# B&R Automation Studio project Embraco_LinkaNaOdlievanieRotorov_DokoncovaciaStanica_Rev2 (part 5)

#### Main.st - Init, cyclic, exit code
```iecst
PROGRAM _INIT
	MpRecipeXml_1.Load:= TRUE;
	ZvolenyUzivatel:= '';
	ZvolenaUroven:= 0;
	TP_ZobrazPopUpPrihlasenie:=1;

END_PROGRAM

PROGRAM _CYCLIC

	//Volanie funkcie SequenceControl//
	SequenceControl(SC:= SC_Uzivatelia);

	//Načítanie receptur z pamäte//
	IF MpRecipeXml_1.Load AND (MpRecipeXml_1.CommandDone OR MpRecipeXml_1.Error) THEN
		MpRecipeXml_1.Load:= FALSE;
		old_a:= 1;
		i:= 0;
		IndexZoznam:= 0;
	END_IF

	//Konfigurácia receptur//
	MpRecipeXml_1.MpLink:= ADR(gRecipeUzivatelXmlLink);  //takto sa menuje mapp komponenta v configurating view//
	MpRecipeXml_1.Enable:= TRUE;
	MpRecipeXml_1.Category:= ADR('UZIVATELIA');
	MpRecipeXml_1.Category:= ADR(strCategory);
	MpRecipeXml_1.DeviceName:= ADR('HDD');  //Názov media, kde sa budú receptury ukladat//
	MpRecipeXml_1.FileName:= ADR('UlozenyUzivatel'); //Názov súboru do ktorého sa receptúry uložia//
	MpRecipeXml_1();

	MpRecipeRegPar_1.MpLink:= ADR(gRecipeUzivatelXmlLink);
	MpRecipeRegPar_1.Enable:= TRUE;
	MpRecipeRegPar_1.Category:= ADR('UZIVATELIA');
	MpRecipeRegPar_1.PVName:= ADR('Uzivatel'); //Názov premenné, kde je vytvorená štruktura dat pre receptury//
	MpRecipeRegPar_1();

	//Zobrazenie názvou receptúr//
	FOR IndexZoznam:=0 TO 20 BY 1 DO
		ZoznamUzivatelov[IndexZoznam]:= Uzivatel[IndexZoznam].Meno;
	END_FOR

	//Posun indexu//
	IF MoveUP THEN
		IF i< 20 THEN
			i:= i+1;
		END_IF
		MoveUP:= FALSE;
	END_IF

	IF MoveDown THEN
		IF i>0 THEN
			i:= i-1;
		END_IF
		MoveDown:= FALSE;
	END_IF

	//Listovanie v uložených uživateloch//
	IF old_a <> i AND i >= 0 AND i <= 20 THEN
		MenoUzivatela:= Uzivatel[i].Meno;
		HesloUzivatela:= Uzivatel[i].Heslo;
		UrovenUzivatela:= Uzivatel[i].UrovenUzivatela;
		old_a:= i;
	END_IF

	//Prihlasovanie//
	CASE SC_Uzivatelia.Step OF

		0://Vynulovanie uživatela//
			SC_Uzivatelia.StepName:= '0 - Nulovanie';
			UlozUzivatelov:= FALSE;
			PrihlasUzivatela:= FALSE;
			VymazUzivatela:= FALSE;
			OdhlasUzivatela:= FALSE;
			MpRecipeXml_1.Save:= FALSE;
			b:= 0;
			SC_Uzivatelia.ResetStep:= TRUE;
			SC_Uzivatelia.Step:= 1;

		1://Rozhodnutie o činnosti//
			SC_Uzivatelia.StepName:= '1 - Rozhodnutie o cinnosti';
			IF UlozUzivatelov THEN
				SC_Uzivatelia.Step:= 10;
			ELSIF PrihlasUzivatela THEN
				SC_Uzivatelia.Step:= 20;
			ELSIF OdhlasUzivatela THEN
				SC_Uzivatelia.Step:= 30;
			ELSIF VymazUzivatela THEN
				SC_Uzivatelia.Step:= 40;
			END_IF

		10://Ulozenie uzivatela//
			SC_Uzivatelia.StepName:= '10 - Ulozenie uzivatela';
			Uzivatel[i].Meno:= MenoUzivatela;
			Uzivatel[i].Heslo:= HesloUzivatela;
			Uzivatel[i].UrovenUzivatela:= UrovenUzivatela;
			MpRecipeXml_1.Save:= TRUE;
			IF MpRecipeXml_1.CommandDone THEN
				SC_Uzivatelia.ResetStep:= TRUE;
				SC_Uzivatelia.Step:= 0;
			END_IF

		20://Čakanie na prihlásenie uživatela//
			SC_Uzivatelia.StepName:= '20 - Kontrola prazdneho uzivatela';
			IF ZadaneMenoUzivatela <> '' AND ZadaneHesloUzivatela <> '' THEN
				SC_Uzivatelia.ResetStep:= TRUE;
				SC_Uzivatelia.Step:= 21;
			ELSE
				ZadaneHesloUzivatela:= '';
				SC_Uzivatelia.ResetStep:= TRUE;
				SC_Uzivatelia.Step:= 0;
			END_IF

		21://Kontrola prihláseného uživatela//
			SC_Uzivatelia.StepName:= '21 - Kontrola prihláseného uzivatela';
			IF Uzivatel[b].Meno = ZadaneMenoUzivatela AND Uzivatel[b].Heslo = ZadaneHesloUzivatela THEN
				ZvolenyUzivatel:= Uzivatel[b].Meno;
				ZvolenaUroven:= Uzivatel[b].UrovenUzivatela;
				ZadaneHesloUzivatela:= '';
				SC_Uzivatelia.ResetStep:= TRUE;
				SC_Uzivatelia.Step:= 0;
			ELSE
				b:= b + 1;
				IF b = 21 OR b < 0 OR b > 21 THEN
					ZadaneMenoUzivatela:= '';
					ZadaneHesloUzivatela:= '';
					SC_Uzivatelia.ResetStep:= TRUE;
					SC_Uzivatelia.Step:= 0;
				END_IF
			END_IF

		30://Odhlásenie uživatela//
			SC_Uzivatelia.StepName:= '30 - Odhlasenie uzivatela';
			ZvolenyUzivatel:= '';
			ZvolenaUroven:= 0;
			SC_Uzivatelia.ResetStep:= TRUE;
			SC_Uzivatelia.Step:= 0;

		40://Vymazanie uživatela//
			SC_Uzivatelia.StepName:= '40 - Vymazanie uzivatela';
			Uzivatel[i].Meno:= '';
			Uzivatel[i].Heslo:= '';
			Uzivatel[i].UrovenUzivatela:= 0;
			MpRecipeXml_1.Save:= TRUE;
			IF MpRecipeXml_1.CommandDone THEN
				SC_Uzivatelia.ResetStep:= TRUE;
				SC_Uzivatelia.Step:= 0;
			END_IF

	END_CASE

END_PROGRAM

PROGRAM _EXIT
	(* Insert code here *)

END_PROGRAM
```

#### Variables.var - Local variables
```iecst
VAR
	strCategory : STRING[80];
	MpRecipeUI_1 : MpRecipeUI;
	UISetup : MpRecipeUISetupType;
	UIConnect : MpRecipeUIConnectType := (0);
	i : INT := 0;
	a : INT;
	old_a : INT := 0;
	MoveUP : BOOL;
	MoveDown : BOOL;
	IndexZoznam : INT;
	b : INT;
END_VAR
```

### Program Logical/Blikace/Blikanie1s (IEC)

#### Blikanie1s.st - Init, cyclic, exit code
```iecst
PROGRAM _INIT
	(* Insert code here *)

END_PROGRAM

PROGRAM _CYCLIC
	IF NOT Blikac1s THEN
		Blikac1s:= TRUE;
	ELSE
		Blikac1s:= FALSE;
	END_IF

END_PROGRAM

PROGRAM _EXIT
	(* Insert code here *)

END_PROGRAM
```

### Program Logical/Blikace/Blikanie200ms (IEC)

#### Blikanie200ms.st - Init, cyclic, exit code
```iecst
PROGRAM _INIT
	(* Insert code here *)

END_PROGRAM

PROGRAM _CYCLIC

	IF NOT Blikac200ms THEN
		Blikac200ms:= TRUE;
	ELSE
		Blikac200ms:= FALSE;
	END_IF

END_PROGRAM

PROGRAM _EXIT
	(* Insert code here *)

END_PROGRAM
```

### Program Logical/Blikace/Blikanie10ms (IEC)

#### Blikanie10ms.st - Init, cyclic, exit code
```iecst
PROGRAM _INIT
	(* Insert code here *)

END_PROGRAM

PROGRAM _CYCLIC
	IF NOT Blikac10ms THEN
		Blikac10ms:= TRUE;
	ELSE
		Blikac10ms:= FALSE;
	END_IF

END_PROGRAM

PROGRAM _EXIT
	(* Insert code here *)

END_PROGRAM
```

### Program Logical/Blikace/Blikanie50ms (IEC)

#### Blikanie50ms.st - Init, cyclic, exit code
```iecst
PROGRAM _INIT
	(* Insert code here *)

END_PROGRAM

PROGRAM _CYCLIC
	IF NOT Blikac50ms THEN
		Blikac50ms:= TRUE;
	ELSE
		Blikac50ms:= FALSE;
	END_IF

END_PROGRAM

PROGRAM _EXIT
	(* Insert code here *)

END_PROGRAM
```

### Program Logical/Blikace/Blikanie500ms (IEC)

#### Blikanie500ms.st - Init, cyclic, exit code
```iecst
PROGRAM _INIT
	(* Insert code here *)

END_PROGRAM

PROGRAM _CYCLIC
	IF NOT Blikac500ms THEN
		Blikac500ms:= TRUE;
	ELSE
		Blikac500ms:= FALSE;
	END_IF

END_PROGRAM

PROGRAM _EXIT
	(* Insert code here *)

END_PROGRAM
```

### Program Logical/Blikace/Blikanie5s (IEC)

#### Blikanie5s.st - Init, cyclic, exit code
```iecst
PROGRAM _INIT
	(* Insert code here *)

END_PROGRAM

PROGRAM _CYCLIC
	IF NOT Blikac5s THEN
		Blikac5s:= TRUE;
	ELSE
		Blikac5s:= FALSE;
	END_IF

END_PROGRAM

PROGRAM _EXIT
	(* Insert code here *)

END_PROGRAM
```

### Program Logical/Receptury/Receptury (IEC)

#### Main.st - Init, cyclic, exit code
```iecst
PROGRAM _INIT

	MpRecipeXml_0.Load:= TRUE;

END_PROGRAM

PROGRAM _CYCLIC

	//Načítanie receptur z pamäte//
	IF MpRecipeXml_0.Load AND (MpRecipeXml_0.CommandDone OR MpRecipeXml_0.Error) THEN
		MpRecipeXml_0.Load:= FALSE;
		old_i:= 1;
		i:= 0;
		IndexZoznam:= 0;
	END_IF

	//Konfigurácia receptur//
	MpRecipeXml_0.MpLink:= ADR(gRecipeXmlLink);  //takto sa menuje mapp komponenta v configurating view//
	MpRecipeXml_0.Enable:= TRUE;
	MpRecipeXml_0.Category:= ADR('RECEPTURY');
	MpRecipeXml_0.DeviceName:= ADR('HDD');  //Názov media, kde sa budú receptury ukladat//
	MpRecipeXml_0.FileName:= ADR('UlozeneReceptury'); //Názov súboru do ktorého sa receptúry uložia//
	MpRecipeXml_0();

	MpRecipeRegPar_0.MpLink:= ADR(gRecipeXmlLink);
	MpRecipeRegPar_0.Enable:= TRUE;
	MpRecipeRegPar_0.Category:= ADR('RECEPTURY');
	MpRecipeRegPar_0.PVName:= ADR('Receptura'); //Názov premenné, kde je vytvorená štruktura dat pre receptury//
	MpRecipeRegPar_0();

	//Zobrazenie názvou receptúr//
	FOR IndexZoznam:=0 TO 20 BY 1 DO
		ZoznamReceptur[IndexZoznam]:= Receptura[IndexZoznam].Nazov;
	END_FOR

	//Posun indexu//
	IF MoveUP THEN
		IF i< 20 THEN
			i:= i+1;
		END_IF
		MoveUP:= FALSE;
	END_IF

	IF MoveDown THEN
		IF i>0 THEN
			i:= i-1;
		END_IF
		MoveDown:= FALSE;
	END_IF

	//Listovanie v uložených recepturach//
	IF old_i <> i THEN
		Nazov:= Receptura[i].Nazov;
		Premenna_1:= Receptura[i].Premenna_1;
		Premenna_2:= Receptura[i].Premenna_2;
		Premenna_3:= Receptura[i].Premenna_3;
		Premenna_4:= Receptura[i].Premenna_4;
		Premenna_5:= Receptura[i].Premenna_5;
		Premenna_6:= Receptura[i].Premenna_6;
		old_i:= i;
	END_IF

	//Uloženie receptury//
	IF UlozRecepturu THEN
		Receptura[i].Nazov:= Nazov;
		Receptura[i].Premenna_1:= Premenna_1;
		Receptura[i].Premenna_2:= Premenna_2;
		Receptura[i].Premenna_3:= Premenna_3;
		Receptura[i].Premenna_4:= Premenna_4;
		Receptura[i].Premenna_5:= Premenna_5;
		Receptura[i].Premenna_6:= Premenna_6;
		MpRecipeXml_0.Save:= TRUE;
		IF MpRecipeXml_0.CommandDone THEN
			MpRecipeXml_0.Save:= FALSE;
			UlozRecepturu:= FALSE;
		END_IF
	END_IF

	//Načitanie receptur do premenných//
	IF NacitajRecepturu THEN
		ZvolenyNazovProduktu:= Nazov;
		ZvolenaPremenna_1:= Premenna_1;
		ZvolenaPremenna_2:= Premenna_2;
		ZvolenaPremenna_3:= Premenna_3;
		ZvolenaPremenna_4:= Premenna_4;
		ZvolenaPremenna_5:= Premenna_5;
		ZvolenaPremenna_6:= Premenna_6;
		NacitajRecepturu:= FALSE;
	END_IF

END_PROGRAM

PROGRAM _EXIT
	(* Insert code here *)

END_PROGRAM
```

#### Variables.var - Local variables
```iecst
VAR
	MpRecipeUI_0 : MpRecipeUI;
	UISetup : MpRecipeUISetupType;
	UIConnect : MpRecipeUIConnectType := (0);
	i : UINT;
	old_i : UINT;
	ZoznamReceptur : ARRAY[0..20] OF STRING[30] := [21('')];
	IndexZoznam : UINT;
	MoveUP : BOOL;
	MoveDown : BOOL;
END_VAR
```

### Program Logical/RiadenieMenicov/RiadenieMenicov (IEC)

#### InverterBasic.st - Program implementation
```iecst
PROGRAM _INIT

	//Nastavenie node number (adresy) na FM P74, DRI -> COnF -> FULL -> COM -> Cbd -> AdrC {0..239] a dlhsie podrzat otocne tlacidlo
	// + OFF/ON menica

	(*Specify your inverter*)
	FM_Menic[1].Input.InverterName	:= 'Meranie - otacanie rotora';
	FM_Menic[1].Input.DeviceString	:= 'IF1.ST2';
	FM_Menic[1].Input.InverterType := P74;
	FM_Menic[1].Input.Node	:= 2; //Rovnaký ako má NOD number menič//

	FM_Menic[2].Input.InverterName	:= 'Valcovanie 1 - otacanie rotora';
	FM_Menic[2].Input.DeviceString	:= 'IF1.ST3';
	FM_Menic[2].Input.InverterType := P74;
	FM_Menic[2].Input.Node	:= 3; //Rovnaký ako má NOD number menič//

	FM_Menic[3].Input.InverterName	:= 'Valcovanie 2 - otacanie nastroja';
	FM_Menic[3].Input.DeviceString	:= 'IF1.ST6';
	FM_Menic[3].Input.InverterType := P74;
	FM_Menic[3].Input.Node	:= 6; //Rovnaký ako má NOD number menič//

	(*X64 error texts for the corresponding error number*)
	ErrorInfo[1].ErrorText[0]	:= '"nOF": No fault code saved';
	ErrorInfo[1].ErrorText[1]	:= '"CFF": Incorrect configuration (parameters)';
	ErrorInfo[1].ErrorText[2]	:= '"CFI": Invalid configuration (parameters)';
	ErrorInfo[1].ErrorText[3]	:= '"SLF": Modbus communication interuption';
	ErrorInfo[1].ErrorText[4]	:= '"ILF": Internal communcation interuption';
	ErrorInfo[1].ErrorText[5]	:= '"CnF": Communication option card';
	ErrorInfo[1].ErrorText[6]	:= '"EPF": External fault';
	ErrorInfo[1].ErrorText[7]	:= '"OCF": Overcurrent';
	ErrorInfo[1].ErrorText[8]	:= '"CrF": Capacitor pre-charge';
	ErrorInfo[1].ErrorText[9]	:= '"LFF": 4 - 20 mA loss';
	ErrorInfo[1].ErrorText[10]	:= '"OHF": Drive overheating';
	ErrorInfo[1].ErrorText[11]	:= '"OLF": Motor overload';
	ErrorInfo[1].ErrorText[12]	:= '"ObF": DC bus overvoltage';
	ErrorInfo[1].ErrorText[13]	:= '"OSF": Line supply overvoltage';
	ErrorInfo[1].ErrorText[14]	:= '"OPF": Motor phase loss';
	ErrorInfo[1].ErrorText[15]	:= '"PHF": Line phase loss';
	ErrorInfo[1].ErrorText[16]	:= '"USF": Line supply undervoltage';
	ErrorInfo[1].ErrorText[17]	:= '"OCF": Motor short-circuit (phase to phase)';
	ErrorInfo[1].ErrorText[18]	:= '"SOF": Motor overspeed';
	ErrorInfo[1].ErrorText[19]	:= '"tnF": Auto-tuning was unsuccessful';
	ErrorInfo[1].ErrorText[20]	:= '"IF1": Unknown rating';
	ErrorInfo[1].ErrorText[21]	:= '"IF2": MMI card';
	ErrorInfo[1].ErrorText[22]	:= '"IF3": MMI communication';
	ErrorInfo[1].ErrorText[23]	:= '"IF4": Industrial EEPROM';
	ErrorInfo[1].ErrorText[24]	:= '"EEF": EEPROM memory';
	ErrorInfo[1].ErrorText[25]	:= '"OCF": Impeding short-circuit';
	ErrorInfo[1].ErrorText[26]	:= '"SCF": Motor short-circuit (to ground)';
	ErrorInfo[1].ErrorText[27]	:= '"OPF": Motor phase loss - 3 phases';
	ErrorInfo[1].ErrorText[28]	:= '"COF": Communication interuption, fault line 2 (CANopen)';
	ErrorInfo[1].ErrorText[29]	:= '"bLF": Brake control';
	ErrorInfo[1].ErrorText[30]	:= '"OCF": Power module, specific to 15kW drives';
	ErrorInfo[1].ErrorText[31]	:= '"SCF": Power module or motor short-circuit, detected at power up.';
	ErrorInfo[1].ErrorText[110]	:= 'Inverter module not Ok';
	(*P74 and P84 error texts for the corresponding error number*)
	ErrorInfo[2].ErrorText[0]	:= '[No fault] (nOF)';
	ErrorInfo[2].ErrorText[1]	:= '[Calibration error] (InF)';
	ErrorInfo[2].ErrorText[2]	:= '[Control Eeprom] (EEF1)';
	ErrorInfo[2].ErrorText[3]	:= '[Incorrect config.] (CFF)';
	ErrorInfo[2].ErrorText[4]	:= '[Invalid config.] (CFI)';
	ErrorInfo[2].ErrorText[5]	:= '[Ground short circuit](SCF3)';
	ErrorInfo[2].ErrorText[6]	:= '[int. com.link] (ILF)';
	ErrorInfo[2].ErrorText[7]	:= '[Com. network] (CnF)';
	ErrorInfo[2].ErrorText[8]	:= '[External flt-LI/Bit] (EPF1)';
	ErrorInfo[2].ErrorText[9]	:= '[Overcurrent] (OCF)';
	ErrorInfo[2].ErrorText[10]	:= '[Precharge] (CrF)';
	ErrorInfo[2].ErrorText[11]	:= '[Speed fdback loss] (SPF)';
	ErrorInfo[2].ErrorText[12]	:= '[Load slipping] (AnF)';
	ErrorInfo[2].ErrorText[13]	:= '[AI2 4-20mA loss] (LFF2)';
	ErrorInfo[2].ErrorText[14]	:= '[PTC1 probe] (PtF1)';
	ErrorInfo[2].ErrorText[15]	:= '[PTC1 overheat] (OtF1)';
	ErrorInfo[2].ErrorText[16]	:= '[Drive overheat] (OHF)';
	ErrorInfo[2].ErrorText[17]	:= '[Motor overload] (OLF)';
	ErrorInfo[2].ErrorText[18]	:= '[Overbraking] (ObF)';
	ErrorInfo[2].ErrorText[19]	:= '[Mains overvoltage] (OSF)';
	ErrorInfo[2].ErrorText[20]	:= '[1 output phase loss] (OPF1)';
	ErrorInfo[2].ErrorText[21]	:= '[Input phase loss] (PHF)';
	ErrorInfo[2].ErrorText[22]	:= '[Undervoltage] (USF)';
	ErrorInfo[2].ErrorText[23]	:= '[Motor short circuit] (SCF1)';
	ErrorInfo[2].ErrorText[24]	:= '[Overspeed] (SOF)';
	ErrorInfo[2].ErrorText[25]	:= '[Auto-tuning] (tnF)';
	ErrorInfo[2].ErrorText[26]	:= '[Rating error] (InF1)';
	ErrorInfo[2].ErrorText[27]	:= '[PWR Calib.] (InF2)';
	ErrorInfo[2].ErrorText[28]	:= '[Int.serial link] (InF3)';
	ErrorInfo[2].ErrorText[29]	:= '[Int.Mfg area] (InF4)';
	ErrorInfo[2].ErrorText[30]	:= '[Power Eeprom] (EEF2)';
	ErrorInfo[2].ErrorText[31]	:= '[Impedant sh. circuit] (SCF2)';
	ErrorInfo[2].ErrorText[32]	:= '[Ground short circuit] (SCF3)';
	ErrorInfo[2].ErrorText[33]	:= '[3out ph loss] (OPF2)';
	ErrorInfo[2].ErrorText[34]	:= '[CAN com.] (COF)';
	ErrorInfo[2].ErrorText[35]	:= '[Brake control] (bLF)';
	ErrorInfo[2].ErrorText[36]	:= '';
	ErrorInfo[2].ErrorText[37]	:= '[Internal-hard init.] (InF7)';
	ErrorInfo[2].ErrorText[38]	:= '[External fault com.] (EPF2)';
	ErrorInfo[2].ErrorText[39]	:= '[Application fault] (APF)';
	ErrorInfo[2].ErrorText[40]	:= '[Internal-ctrl supply] (InF8)';
	ErrorInfo[2].ErrorText[41]	:= '[Brake feedback] (brF)';
	ErrorInfo[2].ErrorText[42]	:= '[PowerSuite com.] (SLF2)';
	ErrorInfo[2].ErrorText[43]	:= '[Enc. coupl.] (ECF)';
	ErrorInfo[2].ErrorText[44]	:= '[Torque/current lim] (SSF)';
	ErrorInfo[2].ErrorText[45]	:= '[HMI com.] (SLF3)';
	ErrorInfo[2].ErrorText[46]	:= '[Power removal] (PrF)';
	ErrorInfo[2].ErrorText[47]	:= '[PTC2 probe] (PtF2)';
	ErrorInfo[2].ErrorText[48]	:= '[PTC2 overheat] (OtF2)';
	ErrorInfo[2].ErrorText[49]	:= '[LI6=PTC probe] (PtFL)';
	ErrorInfo[2].ErrorText[50]	:= '[PTC fault] (OtFL)';
	ErrorInfo[2].ErrorText[51]	:= '[Internal- I measure] (InF9)';
	ErrorInfo[2].ErrorText[52]	:= '[Internal-mains circuit] (InFA)';
	ErrorInfo[2].ErrorText[53]	:= '[Internal- th. sensor] (InFb)';
	ErrorInfo[2].ErrorText[54]	:= '[IGBT overheat] (tJF)';
	ErrorInfo[2].ErrorText[55]	:= '[IGBT short circuit] (SCF4)';
	ErrorInfo[2].ErrorText[56]	:= '[Motor short circuit] (SCF5)';
	ErrorInfo[2].ErrorText[57]	:= '[Torque time-out] (SrF)';
	ErrorInfo[2].ErrorText[58]	:= '[Out. contact. stuck] (FCF1)';
	ErrorInfo[2].ErrorText[59]	:= '[Out. contact. open.] (FCF2)';
	ErrorInfo[2].ErrorText[60]	:= '[Int. T meas.] (InFC)';
	ErrorInfo[2].ErrorText[61]	:= '[AI2 input] (AI2F)';
	ErrorInfo[2].ErrorText[62]	:= '[Encoder] (EnF)';
	ErrorInfo[2].ErrorText[63]	:= '[Thyr. soft charge] (CrF2)';
	ErrorInfo[2].ErrorText[64]	:= '[input contactor] (LCF)';
	ErrorInfo[2].ErrorText[65]	:= '[DB unit sh. circuit] (bUF)';
	ErrorInfo[2].ErrorText[66]	:= '[Diff. I fault] (dCF)';
	ErrorInfo[2].ErrorText[67]	:= '[IGBT desaturation] (HdF)';
	ErrorInfo[2].ErrorText[68]	:= '[Internal-option] (InF6)';
	ErrorInfo[2].ErrorText[69]	:= '[internal- CPU] (InFE)';
	ErrorInfo[2].ErrorText[70]	:= '[BR overload] (bOF)';
	ErrorInfo[2].ErrorText[71]	:= '[AI3 4-20mA loss] (LFF3)';
	ErrorInfo[2].ErrorText[72]	:= '[AI4 4-20mA loss] (LFF4)';
	ErrorInfo[2].ErrorText[73]	:= '[Cards pairing] (HCF)';
	ErrorInfo[2].ErrorText[76]	:= '[Load fault] (dLF)';
	ErrorInfo[2].ErrorText[77]	:= '[Bad conf] (CFI2)';
	ErrorInfo[2].ErrorText[99]	:= '[Ch.sw. fault] (CSF)';
	ErrorInfo[2].ErrorText[100]	:= '[Pr.Underload.Flt] (ULF)';
	ErrorInfo[2].ErrorText[101]	:= '[Proc.Overload Flt] (OLC)';
	ErrorInfo[2].ErrorText[105]	:= '[Angle error] (ASF)';
	ErrorInfo[2].ErrorText[107]	:= '[Safety fault] (SAFF)';
	ErrorInfo[2].ErrorText[108]	:= '[FB fault] (FbE)';
	ErrorInfo[2].ErrorText[109]	:= '[FB stop flt.] (FbES)';
	ErrorInfo[2].ErrorText[110]	:= 'Inverter module not Ok';

END_PROGRAM

PROGRAM _CYCLIC

	//Potvrdenie poruchy pri štarte//
	IF EDGEPOS (BezpOkruhCS_Aktivovany = TRUE) THEN
		FM_Menic[1].Input.Command.Acknowledge:= TRUE;
		FM_Menic[2].Input.Command.Acknowledge:= TRUE;
		FM_Menic[3].Input.Command.Acknowledge:= TRUE;
		CasResetovaniaMenicov.IN:= TRUE;
	END_IF

	IF CasResetovaniaMenicov.Q THEN
		FM_Menic[1].Input.Command.Acknowledge:= FALSE;
		FM_Menic[2].Input.Command.Acknowledge:= FALSE;
		FM_Menic[3].Input.Command.Acknowledge:= FALSE;
		CasResetovaniaMenicov.IN:= FALSE;
	END_IF

	CasResetovaniaMenicov.PT:= T#500ms;
	CasResetovaniaMenicov();

	(*loop trough the number of inverters*)
	FOR InvNr := 1 TO NR_OF_INVERTERS DO

		(************************************(STATUS)************************************)
		FM_Menic[InvNr].Output.Status.Running	:= FM_Menic[InvNr].IO.Running;

		(************************************(ENABLE/DISABLE)************************************)
		IF FM_Menic[InvNr].State = INVERTER_TUNE_X64 OR FM_Menic[InvNr].State = INVERTER_TUNE_P74 OR FM_Menic[InvNr].State = INVERTER_TUNE_P84 THEN
			(*do nothing*)
		ELSE
			(*set the disable voltage and quickstop to the same as module ok*)
			FM_Menic[InvNr].IO.DisableVoltage	:= FM_Menic[InvNr].IO.ModuleOk;
			FM_Menic[InvNr].IO.QuickStop		:= FM_Menic[InvNr].IO.ModuleOk;
		END_IF
		(*********************************(PARAMETER WRITE/READ)*************************************)

		(*Parameters are written trough X2X*)
		IF FM_Menic[InvNr].Input.InverterType = X64 THEN
			(*Tune state also write par to inverter, not at same time*)
			IF FM_Menic[InvNr].State <> INVERTER_TUNE_X64 OR FM_Menic[InvNr].State <> INVERTER_TUNE_P74 OR FM_Menic[InvNr].State <> INVERTER_TUNE_P84 THEN
				(*write acceleration*)
				IF OldAccTime[InvNr] <> FM_Menic[InvNr].Input.AccTime THEN
					AsIOAccWrite_0[InvNr].enable 		:= TRUE;
					AsIOAccWrite_0[InvNr].pChannelName	:= ADR('ACC_Output');
					AsIOAccWrite_0[InvNr].pDeviceName	:= ADR(FM_Menic[InvNr].Input.DeviceString);
					AsIOAccWrite_0[InvNr].value		:= FM_Menic[InvNr].Input.AccTime;
					(*write is done*)
					IF AsIOAccWrite_0[InvNr].status = 0 THEN
						AsIOAccWrite_0[InvNr].enable 	:= FALSE;
						OldAccTime[InvNr]				:= FM_Menic[InvNr].Input.AccTime;
					END_IF
				(*write deceleration*)
				ELSIF OldDecTime[InvNr] <> FM_Menic[InvNr].Input.DecTime THEN
					AsIOAccWrite_0[InvNr].enable 		:= TRUE;
					AsIOAccWrite_0[InvNr].pChannelName	:= ADR('DEC_Output');
					AsIOAccWrite_0[InvNr].pDeviceName	:= ADR(FM_Menic[InvNr].Input.DeviceString);
					AsIOAccWrite_0[InvNr].value		:= FM_Menic[InvNr].Input.DecTime;
					(*write is done*)
					IF AsIOAccWrite_0[InvNr].status = 0 THEN
						AsIOAccWrite_0[InvNr].enable 	:= FALSE;
						OldDecTime[InvNr]				:= FM_Menic[InvNr].Input.DecTime;
					END_IF
				ELSE
					AsIOAccWrite_0[InvNr].enable 	:= FALSE;
				END_IF
			END_IF
		(*Parameters are written trough Powerlink*)
		ELSIF FM_Menic[InvNr].Input.InverterType = P74 OR FM_Menic[InvNr].Input.InverterType = P84 THEN
			(*Tune state also write par to inverter, not at same time*)
			IF FM_Menic[InvNr].State <> INVERTER_TUNE_X64 OR FM_Menic[InvNr].State <> INVERTER_TUNE_P74 OR FM_Menic[InvNr].State <> INVERTER_TUNE_P84 THEN

				EplSDOWrite_0[InvNr].node		:= FM_Menic[InvNr].Input.Node;
				EplSDOWrite_0[InvNr].datalen	:= 2;
				EplSDOWrite_0[InvNr].index		:= 16#203C;
				EplSDOWrite_0[InvNr].pDevice	:= ADR(FM_Menic[InvNr].Input.DeviceString);
				(*write acceleration*)
				IF OldAccTime[InvNr] <> FM_Menic[InvNr].Input.AccTime THEN
					EplSDOWrite_0[InvNr].enable	:= TRUE;
					EplSDOWrite_0[InvNr].pData		:= ADR(FM_Menic[InvNr].Input.AccTime);
					EplSDOWrite_0[InvNr].subindex	:= 2;
					(*write is done*)
					IF EplSDOWrite_0[InvNr].status = 0 THEN
						EplSDOWrite_0[InvNr].enable	:= FALSE;
						OldAccTime[InvNr]				:= FM_Menic[InvNr].Input.AccTime;
					END_IF
				(*write deceleration*)
				ELSIF OldDecTime[InvNr] <> FM_Menic[InvNr].Input.DecTime THEN
					EplSDOWrite_0[InvNr].enable	:= TRUE;
					EplSDOWrite_0[InvNr].pData		:= ADR(FM_Menic[InvNr].Input.DecTime);
					EplSDOWrite_0[InvNr].subindex	:= 3;
					(*write is done*)
					IF EplSDOWrite_0[InvNr].status = 0 THEN
						EplSDOWrite_0[InvNr].enable	:= FALSE;
						OldDecTime[InvNr]				:= FM_Menic[InvNr].Input.DecTime;
					END_IF
				END_IF
			END_IF
		END_IF

		(*********************************(ERROR)*************************************)

		(*Error*)
		IF 	(FM_Menic[InvNr].IO.Fault = TRUE OR FM_Menic[InvNr].IO.ModuleOk = FALSE) AND FM_Menic[InvNr].State <> INVERTER_ERROR THEN
			FM_Menic[InvNr].State := INVERTER_ERROR;
		END_IF

		(*error status*)
		FM_Menic[InvNr].Output.Status.Error	:= FM_Menic[InvNr].IO.Fault;
		FM_Menic[InvNr].Output.Status.ErrorNumber := FM_Menic[InvNr].IO.ErrorNumber;

		(*In case of an inverter fault. Read the error number and select an error text*)
		IF FM_Menic[InvNr].IO.Fault = TRUE OR FM_Menic[InvNr].IO.ModuleOk = FALSE THEN
			IF FM_Menic[InvNr].IO.ModuleOk = TRUE THEN
				(*select list of error text depending on inverter type*)
				IF FM_Menic[InvNr].Input.InverterType = X64 THEN
					FM_Menic[InvNr].Output.Status.ErrorText	:= ErrorInfo[1].ErrorText[FM_Menic[InvNr].IO.ErrorNumber];
				ELSIF FM_Menic[InvNr].Input.InverterType = P74 OR FM_Menic[InvNr].Input.InverterType = P84 THEN
					FM_Menic[InvNr].Output.Status.ErrorText	:= ErrorInfo[2].ErrorText[FM_Menic[InvNr].IO.ErrorNumber];
				END_IF
			ELSIF FM_Menic[InvNr].IO.ModuleOk = FALSE AND FM_Menic[InvNr].IO.ErrorNumber = 0 THEN
				(*Module not okay*)
				FM_Menic[InvNr].Output.Status.ErrorText 	:= ErrorInfo[1].ErrorText[110];
			END_IF
		END_IF

		(************************************(EXTRA FUNCTION)************************************)
		(*Simple brake handling*)
		IF FM_Menic[InvNr].IO.SwitchedOn = TRUE THEN
			FM_Menic[InvNr].IO.Brake := TRUE;
		ELSE
			FM_Menic[InvNr].IO.Brake := FALSE;
		END_IF

		(**************************************************************************************)

		(*Reset substate*)
		IF FM_Menic[InvNr].State <> oldState[InvNr] THEN
			FM_Menic[InvNr].SubState := 0;
			oldState[InvNr] := FM_Menic[InvNr].State;
		END_IF

		CASE FM_Menic[InvNr].State OF

		(**************************************************************************************)

			(*WAIT*)
			INVERTER_WAIT:

				IF FM_Menic[InvNr].Input.Command.RunBackward = TRUE THEN
					FM_Menic[InvNr].IO.Direction 	:= 0;
					FM_Menic[InvNr].State 			:= INVERTER_RUN;
				ELSIF  FM_Menic[InvNr].Input.Command.RunForward = TRUE THEN
					FM_Menic[InvNr].IO.Direction 	:= 1;
					FM_Menic[InvNr].State 			:= INVERTER_RUN;
				ELSIF FM_Menic[InvNr].Input.Command.AutoTune = TRUE THEN
					FM_Menic[InvNr].Input.Command.AutoTune	:= FALSE;
					IF FM_Menic[InvNr].Input.InverterType = X64 THEN
						FM_Menic[InvNr].State 		:= INVERTER_TUNE_X64;
					ELSIF FM_Menic[InvNr].Input.InverterType = P74 THEN
						FM_Menic[InvNr].State 		:= INVERTER_TUNE_P74;
					ELSIF FM_Menic[InvNr].Input.InverterType = P84 THEN
						FM_Menic[InvNr].State 		:= INVERTER_TUNE_P84;
					END_IF
				END_IF;

		(**************************************************************************************)

			INVERTER_TUNE_X64: (*Autotune the inverter*)

				CASE FM_Menic[InvNr].SubState OF

					(**************************************************************************)
					0:	(*make sure to stop the motor*)
						FM_Menic[InvNr].Output.Status.Tuned	:= FALSE;
						FM_Menic[InvNr].IO.Stop				:= TRUE;
						FM_Menic[InvNr].IO.Run					:= FALSE;
						FM_Menic[InvNr].SubState 				:= 10;
					(**************************************************************************)
					10:(*check that it is stopped*)
						IF FM_Menic[InvNr].IO.Running = FALSE THEN
							FM_Menic[InvNr].SubState 	:= 20;
							FM_Menic[InvNr].IO.Stop	:= FALSE;
						END_IF
					(**************************************************************************)
					20:	(*Write tune parameter to inverter X64 through X2X*)
						AsIOAccWrite_0[InvNr].enable 		:= TRUE;
						AsIOAccWrite_0[InvNr].pChannelName	:= ADR('TUN_Output');
						AsIOAccWrite_0[InvNr].pDeviceName	:= ADR(FM_Menic[InvNr].Input.DeviceString);
						AsIOAccWrite_0[InvNr].value			:= 112;

						IF AsIOAccWrite_0[InvNr].status = 0 THEN
							AsIOAccWrite_0[InvNr].enable 	:= FALSE;
							FM_Menic[InvNr].SubState 			:= 30;
						END_IF
					(**************************************************************************)
					30:
						IF FM_Menic[InvNr].IO.ReadyToSwitchOn = TRUE THEN
							FM_Menic[InvNr].IO.SwitchOn	:= TRUE;
							FM_Menic[InvNr].SubState 		:= 40;
						END_IF
					(**************************************************************************)
					40:
						IF FM_Menic[InvNr].IO.SwitchedOn = TRUE THEN
							FM_Menic[InvNr].IO.Run			:= TRUE;
							FM_Menic[InvNr].SubState 		:= 50;
						END_IF
					(**************************************************************************)
					50:	(*Give the tuning some time to be finished*)
						IF FM_Menic[InvNr].IO.Running = TRUE THEN
							TON_TUNE[InvNr].IN :=  TRUE;
							TON_TUNE[InvNr].PT := T#2s;
							IF TON_TUNE[InvNr].Q = TRUE THEN
								TON_TUNE[InvNr].IN 				:= FALSE;
								FM_Menic[InvNr].IO.Run 		:= FALSE;
								FM_Menic[InvNr].SubState 		:= 60;
							END_IF
						END_IF
					(**************************************************************************)
					60:	(*Power off*)
						IF FM_Menic[InvNr].IO.Running = FALSE THEN
							FM_Menic[InvNr].IO.Stop		:= FALSE;
							FM_Menic[InvNr].IO.SwitchOn 	:= FALSE;
							FM_Menic[InvNr].IO.Run 		:= FALSE;
							IF FM_Menic[InvNr].IO.SwitchedOn = FALSE THEN
								FM_Menic[InvNr].Output.Status.Tuned	:= TRUE;
								FM_Menic[InvNr].State 					:= INVERTER_WAIT;
							END_IF
						END_IF
				END_CASE
		(**************************************************************************************)

			INVERTER_TUNE_P74: (*Autotune the inverter*)

				CASE FM_Menic[InvNr].SubState OF

					(**************************************************************************)
					0:	(*make sure to stop the motor and disable voltage*)
						FM_Menic[InvNr].Output.Status.Tuned	:= FALSE;
						FM_Menic[InvNr].IO.Stop				:= TRUE;
						FM_Menic[InvNr].IO.DisableVoltage		:= FALSE;
						FM_Menic[InvNr].IO.QuickStop			:= FALSE;
						FM_Menic[InvNr].SubState 				:= 10;

					(**************************************************************************)
					10:(*check that voltage is disabled*)
						IF FM_Menic[InvNr].IO.SwitchOnDisabled = TRUE AND FM_Menic[InvNr].IO.VoltageEnabled = TRUE THEN
							FM_Menic[InvNr].SubState 			:= 20;
							FM_Menic[InvNr].IO.DisableVoltage	:= TRUE;
							FM_Menic[InvNr].IO.QuickStop		:= TRUE;
						END_IF
					(**************************************************************************)
					20:(*switch controller on*)
						IF FM_Menic[InvNr].IO.SwitchedOn = FALSE AND FM_Menic[InvNr].IO.ReadyToSwitchOn = TRUE THEN
							FM_Menic[InvNr].IO.SwitchOn		:= TRUE;
							FM_Menic[InvNr].IO.Run				:= TRUE;
							FM_Menic[InvNr].SubState 			:= 30;
						END_IF
					(**************************************************************************)
					30:(*check if controller is on*)
						IF FM_Menic[InvNr].IO.SwitchedOn = TRUE AND FM_Menic[InvNr].IO.Running THEN
							FM_Menic[InvNr].SubState 		:= 40;
						END_IF
					(**************************************************************************)
					40:	(*Write tune parameter to inverter P74 or P84 through Powerlink*)
						data := 1;
						EplSDOWrite_0[InvNr].enable	:= TRUE;
						EplSDOWrite_0[InvNr].node		:= FM_Menic[InvNr].Input.Node;
						EplSDOWrite_0[InvNr].datalen	:= 2;
						EplSDOWrite_0[InvNr].index		:= 16#2042;
						EplSDOWrite_0[InvNr].pDevice	:= ADR(FM_Menic[InvNr].Input.DeviceString);
						EplSDOWrite_0[InvNr].pData		:= ADR(data);
						EplSDOWrite_0[InvNr].subindex	:= 9;

						IF EplSDOWrite_0[InvNr].status = 0 THEN
							EplSDOWrite_0[InvNr].enable	:= FALSE;
							FM_Menic[InvNr].SubState 	:= 50;
						END_IF
					(**************************************************************************)
					50:(*Check tuning status*)
						EplSDORead_0[InvNr].enable 		:= TRUE;
						EplSDORead_0[InvNr].pDevice 	:= ADR(FM_Menic[InvNr].Input.DeviceString);
						EplSDORead_0[InvNr].node		:= FM_Menic[InvNr].Input.Node;

						EplSDORead_0[InvNr].datalen		:= SIZEOF(INT);
						EplSDORead_0[InvNr].index		:= 16#2042;
						EplSDORead_0[InvNr].subindex	:= 16#0A;
						EplSDORead_0[InvNr].pData		:= ADR(tuningStatus[InvNr]);

						FM_Menic[InvNr].SubState := 60;
					(**************************************************************************)
					60:	(*if status is wrong return to previus state and try again*)
						IF EplSDORead_0[InvNr].status = 0 THEN
							EplSDORead_0[InvNr].enable := FALSE;
							IF (tuningStatus[InvNr] <> 4) THEN
								FM_Menic[InvNr].SubState := 50;
							ELSE
								paramIndex := 0;
								FM_Menic[InvNr].SubState := 70;
							END_IF
						END_IF
					(**************************************************************************)
					70:	(*Give the tuning some time to be finished*)
						IF FM_Menic[InvNr].IO.Running = TRUE THEN
							TON_TUNE[InvNr].IN :=  TRUE;
							TON_TUNE[InvNr].PT := T#2s;
							IF TON_TUNE[InvNr].Q = TRUE THEN
								TON_TUNE[InvNr].IN 				:= FALSE;
								FM_Menic[InvNr].IO.Run 		:= FALSE;
								FM_Menic[InvNr].SubState 		:= 80;
							END_IF
						END_IF
					(**************************************************************************)
					80:	(*Power off*)
						IF FM_Menic[InvNr].IO.Running = FALSE THEN
							FM_Menic[InvNr].IO.Stop		:= FALSE;
							FM_Menic[InvNr].IO.SwitchOn 	:= FALSE;
							FM_Menic[InvNr].IO.Run 		:= FALSE;
							IF FM_Menic[InvNr].IO.SwitchedOn = FALSE THEN
								FM_Menic[InvNr].Output.Status.Tuned	:= TRUE;
								FM_Menic[InvNr].State 					:= INVERTER_WAIT;
							END_IF
						END_IF
				END_CASE

		(**************************************************************************************)

			INVERTER_TUNE_P84: (*Autotune the inverter*)

				CASE FM_Menic[InvNr].SubState OF

					(**************************************************************************)
					0:	(*make sure to stop the motor and disable voltage*)
						FM_Menic[InvNr].Output.Status.Tuned	:= FALSE;
						FM_Menic[InvNr].IO.Stop				:= TRUE;
						FM_Menic[InvNr].IO.Run					:= FALSE;
						FM_Menic[InvNr].SubState 				:= 10;
					(**************************************************************************)
					10:(*check that it is stopped*)
						IF FM_Menic[InvNr].IO.Running = FALSE THEN
							FM_Menic[InvNr].IO.Stop				:= FALSE;
							FM_Menic[InvNr].SubState 				:= 20;
						END_IF
					(**************************************************************************)
					20:	(*Write tune parameter to inverter P84 through Powerlink*)
						data := 1;
						EplSDOWrite_0[InvNr].enable	:= TRUE;
						EplSDOWrite_0[InvNr].node		:= FM_Menic[InvNr].Input.Node;
						EplSDOWrite_0[InvNr].datalen	:= 2;
						EplSDOWrite_0[InvNr].index		:= 16#2042;
						EplSDOWrite_0[InvNr].pDevice	:= ADR(FM_Menic[InvNr].Input.DeviceString);
						EplSDOWrite_0[InvNr].pData		:= ADR(data);
						EplSDOWrite_0[InvNr].subindex	:= 9;

						IF EplSDOWrite_0[InvNr].status = 0 THEN
							EplSDOWrite_0[InvNr].enable	:= FALSE;
							FM_Menic[InvNr].SubState 	:= 30;
						END_IF
					(**************************************************************************)
					30:(*power on*)
						FM_Menic[InvNr].IO.SwitchOn			:= TRUE;
						FM_Menic[InvNr].IO.Run					:= TRUE;
						FM_Menic[InvNr].IO.SpeedSetpoint		:= 0;

						IF FM_Menic[InvNr].IO.SwitchedOn = TRUE AND FM_Menic[InvNr].IO.Running = TRUE THEN
							FM_Menic[InvNr].SubState 				:= 40;
						END_IF
					(**************************************************************************)
					40:(*Check tuning status*)
						EplSDORead_0[InvNr].enable 		:= TRUE;
						EplSDORead_0[InvNr].pDevice 	:= ADR(FM_Menic[InvNr].Input.DeviceString);
						EplSDORead_0[InvNr].node		:= FM_Menic[InvNr].Input.Node;

						EplSDORead_0[InvNr].datalen		:= SIZEOF(INT);
						EplSDORead_0[InvNr].index		:= 16#2042;
						EplSDORead_0[InvNr].subindex	:= 16#0A;
						EplSDORead_0[InvNr].pData		:= ADR(tuningStatus[InvNr]);

						FM_Menic[InvNr].SubState := 50;
					(**************************************************************************)
					50:	(*if status is wrong return to previus state and try again*)
						IF EplSDORead_0[InvNr].status = 0 THEN
							EplSDORead_0[InvNr].enable := FALSE;

							IF (tuningStatus[InvNr] <> 4) THEN
								FM_Menic[InvNr].SubState := 40;
							ELSE
								paramIndex := 0;
								FM_Menic[InvNr].SubState := 60;
							END_IF
						END_IF
					(**************************************************************************)
					60:	(*Give the tuning some time to be finished*)
						IF FM_Menic[InvNr].IO.Running = TRUE THEN
							TON_TUNE[InvNr].IN :=  TRUE;
							TON_TUNE[InvNr].PT := T#2s;
							IF TON_TUNE[InvNr].Q = TRUE THEN
								TON_TUNE[InvNr].IN 				:= FALSE;
								FM_Menic[InvNr].IO.Run 		:= FALSE;
								FM_Menic[InvNr].SubState 		:= 70;
							END_IF
						END_IF
					(**************************************************************************)
					70:	(*Power off*)
						IF FM_Menic[InvNr].IO.Running = FALSE THEN
							FM_Menic[InvNr].IO.Stop		:= FALSE;
							FM_Menic[InvNr].IO.SwitchOn 	:= FALSE;
							FM_Menic[InvNr].IO.Run 		:= FALSE;
							IF FM_Menic[InvNr].IO.SwitchedOn = FALSE THEN
								FM_Menic[InvNr].Output.Status.Tuned	:= TRUE;
								FM_Menic[InvNr].State 					:= INVERTER_WAIT;
							END_IF
						END_IF
				END_CASE
		(**************************************************************************************)

			(*RUN*)
			INVERTER_RUN:

				(*Swith on and run*)
				IF FM_Menic[InvNr].IO.ReadyToSwitchOn THEN
					FM_Menic[InvNr].IO.SwitchOn := TRUE;
					IF FM_Menic[InvNr].IO.SwitchedOn THEN
						FM_Menic[InvNr].IO.Run := TRUE;
					END_IF
				END_IF

				(*Select speed*)
				IF FM_Menic[InvNr].Input.Command.RunLowSpeed = TRUE THEN
					FM_Menic[InvNr].IO.SpeedSetpoint := FM_Menic[InvNr].Input.LowSpeed;
				ELSE
					FM_Menic[InvNr].IO.SpeedSetpoint := FM_Menic[InvNr].Input.HighSpeed;
				END_IF

				(*Stop when comand is false*)
				IF FM_Menic[InvNr].IO.Direction = 0 AND FM_Menic[InvNr].Input.Command.RunBackward = FALSE THEN
					FM_Menic[InvNr].State 				:= INVERTER_STOP;
				ELSIF FM_Menic[InvNr].IO.Direction = 1 AND FM_Menic[InvNr].Input.Command.RunForward = FALSE THEN
					FM_Menic[InvNr].State 				:= INVERTER_STOP;
				END_IF;

		(**************************************************************************************)

			INVERTER_STOP:(*STOP*)

				CASE FM_Menic[InvNr].SubState OF

					0:
						(*stop command bit*)
						IF FM_Menic[InvNr].Input.StopType = 0 THEN
							FM_Menic[InvNr].SubState := 10;
						(*freeweel stop*)
						ELSIF FM_Menic[InvNr].Input.StopType = 1 THEN
							FM_Menic[InvNr].SubState := 20;
						END_IF
					(**************************************************************************)
					10:
						(*check standstill*)
						FM_Menic[InvNr].IO.Stop 			:= TRUE;
						FM_Menic[InvNr].IO.Run				:= TRUE;
						FM_Menic[InvNr].IO.SpeedSetpoint	:= 0;

						IF FM_Menic[InvNr].IO.SpeedMode = FALSE AND FM_Menic[InvNr].IO.OutputFrequency = 0 AND FM_Menic[InvNr].IO.MotorTorque = 0 AND FM_Menic[InvNr].IO.MotorCurrent = 0 THEN
							FM_Menic[InvNr].IO.Stop 		:= FALSE;
							FM_Menic[InvNr].IO.Run			:= FALSE;
							FM_Menic[InvNr].State 			:= INVERTER_POWER_OFF;
						END_IF
					(**************************************************************************)
					20:
						(*set run command off*)
						FM_Menic[InvNr].IO.Run				:= FALSE;
						FM_Menic[InvNr].IO.SpeedSetpoint	:= 0;

						IF FM_Menic[InvNr].IO.SpeedMode = FALSE AND FM_Menic[InvNr].IO.OutputFrequency = 0 AND FM_Menic[InvNr].IO.MotorTorque = 0 AND FM_Menic[InvNr].IO.MotorCurrent = 0 THEN
							FM_Menic[InvNr].IO.Stop 		:= FALSE;
							FM_Menic[InvNr].State 			:= INVERTER_POWER_OFF;
						END_IF
				END_CASE

	(**************************************************************************************)

			INVERTER_POWER_OFF:	(*POWER OFF*)

				(*set comand bits to inverter*)
				FM_Menic[InvNr].IO.Run			:= FALSE;
				FM_Menic[InvNr].IO.SwitchOn 	:= FALSE;

				(*exit state on status*)
				IF FM_Menic[InvNr].IO.SwitchedOn = FALSE THEN
					FM_Menic[InvNr].State 				:= INVERTER_WAIT;
				END_IF

	(**************************************************************************************)

			INVERTER_ERROR:	(*ERROR*)

				(*reset fault by comand bit. A hardware reset through an assigned DI might be required*)
				IF FM_Menic[InvNr].Input.Command.Acknowledge = TRUE THEN
					FM_Menic[InvNr].IO.FaultReset := TRUE;
				END_IF

				(*Set the run commands to false*)
				FM_Menic[InvNr].Input.Command.RunForward	:= FALSE;
				FM_Menic[InvNr].Input.Command.RunBackward	:= FALSE;

				(*make sure inverter is stopped*)
				FM_Menic[InvNr].IO.Run			:= FALSE;
				FM_Menic[InvNr].IO.Stop		:= FALSE;
				FM_Menic[InvNr].IO.SwitchOn	:= FALSE;

				(*exit state if there is no fault*)
				IF FM_Menic[InvNr].IO.Fault = FALSE AND FM_Menic[InvNr].IO.ReadyToSwitchOn = TRUE THEN
					FM_Menic[InvNr].IO.FaultReset 				:= FALSE;
					FM_Menic[InvNr].Input.Command.Acknowledge 	:= FALSE;
					FM_Menic[InvNr].Output.Status.ErrorText	:= '';
					FM_Menic[InvNr].Output.Status.ErrorNumber	:= 0;
					FM_Menic[InvNr].State						:= INVERTER_WAIT;
				END_IF

			END_CASE;

	(**************************************************************************************)

		(*FUB calls*)
		EplSDOWrite_0[InvNr]();
		AsIOAccWrite_0[InvNr]();
		EplSDORead_0[InvNr]();
		TON_TUNE[InvNr]();

	END_FOR

END_PROGRAM

PROGRAM _EXIT

END_PROGRAM
```

#### InverterBasic.var - Local variables
```iecst
VAR
	oldState : ARRAY[1..NR_OF_INVERTERS] OF INVERTER_STATES;
	AsIOAccWrite_0 : ARRAY[1..NR_OF_INVERTERS] OF AsIOAccWrite;
	TON_TUNE : ARRAY[1..NR_OF_INVERTERS] OF TON;
	OldAccTime : ARRAY[1..NR_OF_INVERTERS] OF UINT;
	OldDecTime : ARRAY[1..NR_OF_INVERTERS] OF UINT;
	EplSDOWrite_0 : ARRAY[1..NR_OF_INVERTERS] OF EplSDOWrite;
	data : INT;
	InvNr : USINT;
	EplSDORead_0 : ARRAY[0..NR_OF_INVERTERS] OF EplSDORead;
	paramIndex : USINT;
	tuningStatus : ARRAY[0..NR_OF_INVERTERS] OF INT;
	CasResetovaniaMenicov : TON;
END_VAR
```

### Package Logical/RiadenieServ/VstupnyManipulator - Vstupny manipulator

### Data object Logical/RiadenieServ/VstupnyManipulator/gAxis01a (Apt)

#### gAxis01a.apt
```
AcoposParameterTable:
  Root Parameters
```

### Data object Logical/RiadenieServ/VstupnyManipulator/gAxis01i (Ax)

#### gAxis01i.ax
```
InitParameter (Version=5.00.2)
  ACP10AXIS_typ:
    dig_in:
      level:
        reference = ncACTIV_HI + ncFORCE
        pos_hw_end = ncACTIV_HI + ncFORCE
        neg_hw_end = ncACTIV_HI + ncFORCE
        trigger1 = ncACTIV_HI
        trigger2 = ncACTIV_HI
    encoder_if:
      parameter:
        count_dir = ncSTANDARD
        scaling:
          load:
            units = 800
            rev_motor = 1
    limit:
      parameter:
        v_pos = 900000.0
        v_neg = 900000.0
        a1_pos = 9.0E+07
        a2_pos = 9.0E+07
        a1_neg = 9.0E+07
        a2_neg = 9.0E+07
        t_jolt = 0.0
        t_in_pos = 0.0
        pos_sw_end = 8388607
        neg_sw_end = -8388608
        ds_warning = 500.0
        ds_stop = 1000.0
        a_stop = 1.0E+30
        dv_stop = 0.0
        dv_stop_mode = ncOFF
    controller:
      mode = ncPOSITION + ncFF
      position:
        kv = 414.0
        tn = 0.0
        t_predict = 0.0004
        t_total = 0.0004
        p_max = 1.0E+30
        i_max = 0.0
      speed:
        kv = 1.75
        tn = 0.0
        t_filter = 0.0
        isq_filter1:
          type = ncOFF
          a0 = 0.0
          a1 = 0.0
          b0 = 0.0
          b1 = 0.0
          b2 = 0.0
          c0_par_id = 0
          c1_par_id = 0
        isq_filter2:
          type = ncOFF
          a0 = 0.0
          a1 = 0.0
          b0 = 0.0
          b1 = 0.0
          b2 = 0.0
          c0_par_id = 0
          c1_par_id = 0
        isq_filter3:
          type = ncOFF
          a0 = 0.0
          a1 = 0.0
          b0 = 0.0
          b1 = 0.0
          b2 = 0.0
          c0_par_id = 0
          c1_par_id = 0
      uf:
        type = ncLINEAR
        auto_config = ncMOTOR_PAR
        u0 = 0.0
        un = 0.0
        fn = 50.0
        k_f_slip = 0.0
      ff:
        torque_load = 0.0
        torque_pos = 0.0227787
        torque_neg = 0.0207411
        kv_torque = 0.00516676
        inertia = 5.89275E-05
        t_filter_a = 0.0
    move:
      stop:
        parameter[0]:
          decel_ramp = ncA_LIMIT
          controller = ncON
        parameter[1]:
          decel_ramp = ncA_LIMIT
          controller = ncON
        parameter[2]:
          decel_ramp = ncA_LIMIT
          controller = ncON
        parameter[3]:
          decel_ramp = ncA_LIMIT
          controller = ncON
        quickstop:
          decel_ramp = ncA_LIMIT
        drive_error:
          decel_ramp = ncA_LIMIT
      homing:
        parameter:
          s = 0
          v_switch = 1500.0
          v_trigger = 500.0
          a = 3000.0
          mode = ncEND_SWITCH
          edge_sw = ncNEGATIVE
          start_dir = ncNEGATIVE
          trigg_dir = ncPOSITIVE
          ref_pulse = ncOFF
          fix_dir = ncOFF
          tr_s_block = 0.0
          torque_lim = 0.0
          ds_block = 0.0
          ds_stop = 0.0
      basis:
        parameter:
          v_pos = 5000.0
          v_neg = 5000.0
          a1_pos = 50000.0
          a2_pos = 50000.0
          a1_neg = 50000.0
          a2_neg = 50000.0
    message:
      text:
        parameter:
          format = ncBREAK
          columns = 80
          data_modul = acp10etxen
```

### Package Logical/RiadenieServ/VystupnyManipulator - Vystupny manipulator

### Data object Logical/RiadenieServ/VystupnyManipulator/gAxis02a (Apt)

#### gAxis02a.apt
```
AcoposParameterTable:
  Root Parameters
```

### Data object Logical/RiadenieServ/VystupnyManipulator/gAxis02i (Ax)

#### gAxis02i.ax
```
InitParameter (Version=5.00.2)
  ACP10AXIS_typ:
    dig_in:
      level:
        reference = ncACTIV_HI + ncFORCE
        pos_hw_end = ncACTIV_HI + ncFORCE
        neg_hw_end = ncACTIV_HI + ncFORCE
        trigger1 = ncACTIV_HI
        trigger2 = ncACTIV_HI
    encoder_if:
      parameter:
        count_dir = ncSTANDARD
        scaling:
          load:
            units = 800
            rev_motor = 1
    limit:
      parameter:
        v_pos = 900000.0
        v_neg = 900000.0
        a1_pos = 9.0E+07
        a2_pos = 9.0E+07
        a1_neg = 9.0E+07
        a2_neg = 9.0E+07
        t_jolt = 0.0
        t_in_pos = 0.0
        pos_sw_end = 8388607
        neg_sw_end = -8388608
        ds_warning = 500.0
        ds_stop = 1000.0
        a_stop = 1.0E+30
        dv_stop = 0.0
        dv_stop_mode = ncOFF
    controller:
      mode = ncPOSITION + ncFF
      position:
        kv = 394.0
        tn = 0.0
        t_predict = 0.0004
        t_total = 0.0004
        p_max = 1.0E+30
        i_max = 0.0
      speed:
        kv = 1.5
        tn = 0.0
        t_filter = 0.0
        isq_filter1:
          type = ncOFF
          a0 = 0.0
          a1 = 0.0
          b0 = 0.0
          b1 = 0.0
          b2 = 0.0
          c0_par_id = 0
          c1_par_id = 0
        isq_filter2:
          type = ncOFF
          a0 = 0.0
          a1 = 0.0
          b0 = 0.0
          b1 = 0.0
          b2 = 0.0
          c0_par_id = 0
          c1_par_id = 0
        isq_filter3:
          type = ncOFF
          a0 = 0.0
          a1 = 0.0
          b0 = 0.0
          b1 = 0.0
          b2 = 0.0
          c0_par_id = 0
          c1_par_id = 0
      uf:
        type = ncLINEAR
        auto_config = ncMOTOR_PAR
        u0 = 0.0
        un = 0.0
        fn = 50.0
        k_f_slip = 0.0
      ff:
        torque_load = 0.0
        torque_pos = 0.00875144
        torque_neg = 0.00666361
        kv_torque = 0.00855945
        inertia = 5.52298E-05
        t_filter_a = 0.0
    move:
      stop:
        parameter[0]:
          decel_ramp = ncA_LIMIT
          controller = ncON
        parameter[1]:
          decel_ramp = ncA_LIMIT
          controller = ncON
        parameter[2]:
          decel_ramp = ncA_LIMIT
          controller = ncON
        parameter[3]:
          decel_ramp = ncA_LIMIT
          controller = ncON
        quickstop:
          decel_ramp = ncA_LIMIT
        drive_error:
          decel_ramp = ncA_LIMIT
      homing:
        parameter:
          s = 0
          v_switch = 1500.0
          v_trigger = 500.0
          a = 3000.0
          mode = ncEND_SWITCH
          edge_sw = ncNEGATIVE
          start_dir = ncNEGATIVE
          trigg_dir = ncPOSITIVE
          ref_pulse = ncOFF
          fix_dir = ncOFF
          tr_s_block = 0.0
          torque_lim = 0.0
          ds_block = 0.0
          ds_stop = 0.0
      basis:
        parameter:
          v_pos = 5000.0
          v_neg = 5000.0
          a1_pos = 50000.0
          a2_pos = 50000.0
          a1_neg = 50000.0
          a2_neg = 50000.0
    message:
      text:
        parameter:
          format = ncBREAK
          columns = 80
          data_modul = acp10etxen
```

### Package Logical/RiadenieServ/ZdvihValcovacky - Zdvih valcovacky_valcovanie 1

### Data object Logical/RiadenieServ/ZdvihValcovacky/gAxis03a (Apt)

#### gAxis03a.apt
```
AcoposParameterTable:
  Root Parameters
```

### Data object Logical/RiadenieServ/ZdvihValcovacky/gAxis03i (Ax)

#### gAxis03i.ax
```
InitParameter (Version=5.00.2)
  ACP10AXIS_typ:
    dig_in:
      level:
        reference = ncACTIV_HI + ncFORCE
        pos_hw_end = ncACTIV_HI + ncFORCE
        neg_hw_end = ncACTIV_HI + ncFORCE
        trigger1 = ncACTIV_HI
        trigger2 = ncACTIV_HI
    encoder_if:
      parameter:
        count_dir = ncSTANDARD
        scaling:
          load:
            units = 1000
            rev_motor = 1
    limit:
      parameter:
        v_pos = 900000.0
        v_neg = 900000.0
        a1_pos = 9.0E+07
        a2_pos = 9.0E+07
        a1_neg = 9.0E+07
        a2_neg = 9.0E+07
        t_jolt = 0.0
        t_in_pos = 0.0
        pos_sw_end = 8388607
        neg_sw_end = -8388608
        ds_warning = 500.0
        ds_stop = 1000.0
        a_stop = 1.0E+30
        dv_stop = 0.0
        dv_stop_mode = ncOFF
    controller:
      mode = ncPOSITION + ncFF
      position:
        kv = 434.0
        tn = 0.0
        t_predict = 0.0004
        t_total = 0.0004
        p_max = 1.0E+30
        i_max = 0.0
      speed:
        kv = 0.95
        tn = 0.0
        t_filter = 0.0
        isq_filter1:
          type = ncOFF
          a0 = 0.0
          a1 = 0.0
          b0 = 0.0
          b1 = 0.0
          b2 = 0.0
          c0_par_id = 0
          c1_par_id = 0
        isq_filter2:
          type = ncOFF
          a0 = 0.0
          a1 = 0.0
          b0 = 0.0
          b1 = 0.0
          b2 = 0.0
          c0_par_id = 0
          c1_par_id = 0
        isq_filter3:
          type = ncOFF
          a0 = 0.0
          a1 = 0.0
          b0 = 0.0
          b1 = 0.0
          b2 = 0.0
          c0_par_id = 0
          c1_par_id = 0
      uf:
        type = ncLINEAR
        auto_config = ncMOTOR_PAR
        u0 = 0.0
        un = 0.0
        fn = 50.0
        k_f_slip = 0.0
      ff:
        torque_load = -0.00177144
        torque_pos = 0.0412463
        torque_neg = 0.039468
        kv_torque = 0.0052849
        inertia = 2.64383E-05
        t_filter_a = 0.0
    move:
      stop:
        parameter[0]:
          decel_ramp = ncA_LIMIT
          controller = ncON
        parameter[1]:
          decel_ramp = ncA_LIMIT
          controller = ncON
        parameter[2]:
          decel_ramp = ncA_LIMIT
          controller = ncON
        parameter[3]:
          decel_ramp = ncA_LIMIT
          controller = ncON
        quickstop:
          decel_ramp = ncA_LIMIT
        drive_error:
          decel_ramp = ncA_LIMIT
      homing:
        parameter:
          s = 0
          v_switch = 1000.0
          v_trigger = 500.0
          a = 3000.0
          mode = ncEND_SWITCH
          edge_sw = ncNEGATIVE
          start_dir = ncNEGATIVE
          trigg_dir = ncPOSITIVE
          ref_pulse = ncOFF
          fix_dir = ncOFF
          tr_s_block = 0.0
          torque_lim = 0.0
          ds_block = 0.0
          ds_stop = 0.0
      basis:
        parameter:
          v_pos = 5000.0
          v_neg = 5000.0
          a1_pos = 50000.0
          a2_pos = 50000.0
          a1_neg = 50000.0
          a2_neg = 50000.0
    message:
      text:
        parameter:
          format = ncBREAK
          columns = 80
          data_modul = acp10etxen
```

### Package Logical/RiadenieServ/ZdvihRotora - Zdvih rotora_valcovanie 2

### Data object Logical/RiadenieServ/ZdvihRotora/gAxis04a (Apt)

#### gAxis04a.apt
```
AcoposParameterTable:
  Root Parameters
```

### Data object Logical/RiadenieServ/ZdvihRotora/gAxis04i (Ax)

#### gAxis04i.ax
```
InitParameter (Version=5.04.1)
  ACP10AXIS_typ:
    dig_in:
      level:
        reference = ncACTIV_HI + ncFORCE
        pos_hw_end = ncACTIV_HI + ncFORCE
        neg_hw_end = ncACTIV_HI + ncFORCE
        trigger1 = ncACTIV_HI
        trigger2 = ncACTIV_HI
    encoder_if:
      parameter:
        count_dir = ncSTANDARD
        scaling:
          load:
            units = 1000
            rev_motor = 1
    limit:
      parameter:
        v_pos = 100000.0
        v_neg = 100000.0
        a1_pos = 5000000.0
        a2_pos = 5000000.0
        a1_neg = 5000000.0
        a2_neg = 5000000.0
        t_jolt = 0.0
        t_in_pos = 0.0
        pos_sw_end = 8388607
        neg_sw_end = -8388608
        ds_warning = 500.0
        ds_stop = 1000.0
        a_stop = 1.0E+30
        dv_stop = 0.0
        dv_stop_mode = ncOFF
    controller:
      mode = ncPOSITION
      position:
        kv = 408.0
        tn = 0.0
        t_predict = 0.0004
        t_total = 0.0004
        p_max = 1.0E+30
        i_max = 0.0
      speed:
        kv = 10.85
        tn = 0.0
        t_filter = 0.0
        isq_filter1:
          type = ncOFF
          a0 = 0.0
          a1 = 0.0
          b0 = 0.0
          b1 = 0.0
          b2 = 0.0
          c0_par_id = 0
          c1_par_id = 0
        isq_filter2:
          type = ncOFF
          a0 = 0.0
          a1 = 0.0
          b0 = 0.0
          b1 = 0.0
          b2 = 0.0
          c0_par_id = 0
          c1_par_id = 0
        isq_filter3:
          type = ncOFF
          a0 = 0.0
          a1 = 0.0
          b0 = 0.0
          b1 = 0.0
          b2 = 0.0
          c0_par_id = 0
          c1_par_id = 0
      uf:
        type = ncLINEAR + ncCORRECTION
        auto_config = ncMOTOR_PAR
        u0 = 0.0
        un = 0.0
        fn = 50.0
        k_f_slip = 0.0
      ff:
        mode = ncSTANDARD
        torque_load = 0.0
        torque_pos = 0.0
        torque_neg = 0.0
        kv_torque = 0.0
        inertia = 0.0
        t_filter_a = 0.0
      fb:
        mode = ncSTANDARD
        speed_mix_ratio = 0.0
        speed_kv = 0.0
      model:
        mass1:
          inertia = 0.0
          viscous_friction = 0.0
        mass2:
          inertia = 0.0
          viscous_friction = 0.0
          stiffness = 0.0
          damping = 0.0
    move:
      stop:
        parameter[0]:
          decel_ramp = ncA_LIMIT
          controller = ncON
        parameter[1]:
          decel_ramp = ncA_LIMIT
          controller = ncON
        parameter[2]:
          decel_ramp = ncA_LIMIT
          controller = ncON
        parameter[3]:
          decel_ramp = ncA_LIMIT
          controller = ncON
        quickstop:
          decel_ramp = ncA_LIMIT
          t_jolt = 0.0
        drive_error:
          decel_ramp = ncA_LIMIT
      homing:
        parameter:
          s = 0
          v_switch = 500.0
          v_trigger = 50.0
          a = 5000.0
          mode = ncEND_SWITCH
          edge_sw = ncNEGATIVE
          start_dir = ncNEGATIVE
          trigg_dir = ncPOSITIVE
          ref_pulse = ncOFF
          fix_dir = ncOFF
          tr_s_block = 0.0
          torque_lim = 0.0
          ds_block = 0.0
          ds_stop = 0.0
      basis:
        parameter:
          v_pos = 200.0
          v_neg = 50.0
          a1_pos = 5000.0
          a2_pos = 5000.0
          a1_neg = 5000.0
          a2_neg = 5000.0
    message:
      text:
        parameter:
          format = ncBREAK
          columns = 80
          data_modul = acp10etxen
```

### Data object Logical/RiadenieServ/acp10etxen (Ett)

- acp10etxen.ett (not shown)

### Program Logical/RiadenieServ/Serva_PriradenieVstupov (IEC)

#### Main.st - Init, cyclic, exit code
```iecst
PROGRAM _INIT
	(* Insert code here *)

END_PROGRAM

PROGRAM _CYCLIC

	//Pojazd vstupného manipulátora//
	Servo1_PriradenieSnimacov.Axis:= ADR(gAxis01);
	Servo1_PriradenieSnimacov.Enable:= TRUE;
	Servo1_PriradenieSnimacov.PosHWSwitch:= diVstupManipul_PrednyLimitSnimac;
	Servo1_PriradenieSnimacov.NegHWSwitch:= diVstupManipul_ZadnyLimitSnimac;
	Servo1_PriradenieSnimacov();

	//Pojazd výstupného manipulátora//
	Servo2_PriradenieSnimacov.Axis:= ADR(gAxis02);
	Servo2_PriradenieSnimacov.Enable:= TRUE;
	Servo2_PriradenieSnimacov.PosHWSwitch:= diVystupManipul_PrednyLimSnimac;
	Servo2_PriradenieSnimacov.NegHWSwitch:= diVystupManipul_ZadnyLimSnimac;
	Servo2_PriradenieSnimacov();

	//Zdvih valcovačky - stanica valcovania 1//
	Servo3_PriradenieSnimacov.Axis:= ADR(gAxis03);
	Servo3_PriradenieSnimacov.Enable:= TRUE;
	Servo3_PriradenieSnimacov.PosHWSwitch:= diValcovanie_SpodnyLimitSnimac;
	Servo3_PriradenieSnimacov.NegHWSwitch:= diValcovanie_HornyLimitSnimac;
	Servo3_PriradenieSnimacov();

	//Zdvih rotora - stanica valcovania 2//
	Servo4_PriradenieSnimacov.Axis:= ADR(gAxis04);
	Servo4_PriradenieSnimacov.Enable:= TRUE;
	Servo4_PriradenieSnimacov.PosHWSwitch:= diValc2_ZdvihHornyLimit;
	Servo4_PriradenieSnimacov.NegHWSwitch:= diValc2_ZdvihSpodnyLimit;
	Servo4_PriradenieSnimacov();

END_PROGRAM

PROGRAM _EXIT
	(* Insert code here *)

END_PROGRAM
```

### Program Logical/RiadenieServ/RiadenieServ (IEC)

#### Main.st - Init, cyclic, exit code
```iecst
PROGRAM _INIT
	Motion[1].par.axis:= ADR(gAxis01);  //Vstupny manipulator//
	Motion[2].par.axis:= ADR(gAxis02);  //Vystupny manipulator//
	Motion[3].par.axis:= ADR(gAxis03);  //Zdvih valcovacky - stanica valcovania 1//
	Motion[4].par.axis:= ADR(gAxis04);  //Zdvih rotora - stanica valcovania 2//

END_PROGRAM

PROGRAM _CYCLIC

	FOR idx:=1 TO MAX_MOTION DO
		Motion[idx].enable := TRUE;
		Motion[idx];
	END_FOR

	IF BezpOkruhCS_Aktivovany THEN
		Motion[1].cmd.power:= TRUE;
		Motion[2].cmd.power:= TRUE;
		Motion[3].cmd.power:= TRUE;
		Motion[4].cmd.power:= TRUE;
	ELSE
		Motion[1].cmd.power:= FALSE;
		Motion[2].cmd.power:= FALSE;
		Motion[3].cmd.power:= FALSE;
		Motion[4].cmd.power:= FALSE;
	END_IF

	IF EDGEPOS (BezpOkruhOplotenia_Aktivovany = TRUE) THEN
		Motion[1].cmd.autoInicialization:= TRUE;
		Motion[2].cmd.autoInicialization:= TRUE;
		Motion[3].cmd.autoInicialization:= TRUE;
		Motion[4].cmd.autoInicialization:= TRUE;
		CasVypnutiaAutoInitServ.IN:= TRUE;
	END_IF
	IF CasVypnutiaAutoInitServ.Q AND Motion[1].errorID = 0 AND Motion[2].errorID = 0 AND Motion[3].errorID = 0 AND Motion[4].errorID = 0  THEN
		Motion[1].cmd.autoInicialization:= FALSE;
		Motion[2].cmd.autoInicialization:= FALSE;
		Motion[3].cmd.autoInicialization:= FALSE;
		Motion[4].cmd.autoInicialization:= FALSE;
		CasVypnutiaAutoInitServ.IN:= FALSE;
	END_IF

	CasVypnutiaAutoInitServ.PT:= T#3s;
	CasVypnutiaAutoInitServ();

	//Stavy homingov serv//
	VstupManipulator_HomingOK:= Motion[1].status.DriveStatus.HomingOk;
	VystupManipulator_HomingOK:= Motion[2].status.DriveStatus.HomingOk;
	Valcovanie_HomingOK:= Motion[3].status.DriveStatus.HomingOk;
	Valcovanie2_HomingOK:= Motion[4].status.DriveStatus.HomingOk;

	//Zobrazenie aktuálnej pozície serv//
	VstupManipulator_AktualPozMM:= (Motion[1].status.ActPosition / 100);
	VystupManipulator_AktualPozMM:= (Motion[2].status.ActPosition / 100);
	Valcovanie_AktualPozMM:= (Motion[3].status.ActPosition / 100);
	Valcovanie2_AktualPozMM:= (Motion[4].status.ActPosition / 100);

	//Stav serva Ready//
	IF Motion[1].errorID = 0 AND Motion[2].errorID = 0 AND Motion[3].errorID = 0 AND Motion[4].errorID = 0 THEN
		Stav_ServaREADY:= TRUE;
	ELSE
		Stav_ServaREADY:= FALSE;
	END_IF

END_PROGRAM

PROGRAM _EXIT
	(* Insert code here *)

END_PROGRAM
```

#### Variables.var - Local variables
```iecst
VAR
	CasVypnutiaAutoInitServ : TON;
END_VAR
```

- Visualisation Logical/Vizualizacia/Visu (not shown)

### Poznamky.txt
```
Heslo do safety - vlmardo
Stanica valcovania 1 - Zdvih valcovačky - 1ot serva = 10mm t.j. 1000 jednotiek
Manipulator - 1ot serva = 8mm  t.j. 800 jednotiek
Stanica valcovania 2 - Zdvih rotora - 1ot serva = 10mm t.j. 1000 jednotiek
```
